FUNCTION_BLOCK PUBLIC FB_StationBase EXTENDS FB_ComponentBase IMPLEMENTS IStation
VAR_INPUT
	/// Enable items
	bEmergencyStopOk 	: BOOL;
	bSafetyOk 			: BOOL;
	bEnable 			: BOOL;
	bAutoHome 			: BOOL;		// if its true station will be homed by start button
	iNumberOfStepChains	: INT := 1;	// count of stepchains per station
	iStepChainIndex		: INT; 		// index to link text of choosed stepchain to hmi
END_VAR
VAR_OUTPUT
	nStateColor			: DWORD;	// color for state of station
	bBusy				: BOOL;		// station is busy
	bTransferEnable		: BOOL;		// transfer enable from station
	stTextAuto			: ST_Text;	// T_MaxString;
	stTextHome			: ST_Text;	// T_MaxString;
	
	/// error-stop status
	bAutoStop_Error		: BOOL;
END_VAR
VAR
	/// Refs
	stHmiToStation		: REFERENCE TO ST_DefaultHmiToPlc;				// default hmi to station
	stHmiManualIn		: REFERENCE TO ST_HMI_BASE_STATION_MANUAL_IN;	// hmi manual to station
	stHmiManualOut		: REFERENCE TO ST_HMI_BASE_STATION_MANUAL_OUT;	// hmi manual from station
	stLocalSettings		: REFERENCE TO ST_StationDynSettings;			// dyn. station settings
	stLocalMonitoring	: REFERENCE TO ST_Monitoring_Station;			// dyn. station monitoring
	
	stLocalSettingsBackup	: ST_StationDynSettings;	// dyn. station settings
	
	/// private var's
	nStationNb		: INT;
	eStation		: E_Station;
	eParent 		: E_Module;
	eOpMode			: E_OpMode;	
	bStopped		: BOOL := TRUE;
	bTipEnable		: BOOL;
	
	/// enable var's
	bRunCycle, bRunStep, 
	bRunHoming, bInHome,
	bEnableManualStep		 : BOOL;

	/// counter
	diCycles				: UDINT; // Zykluszähler
	diLastCycleTime			: UDINT; // letzte Zykluszeit [ms]
	
	tonOpModeOff			: TON;
	fTrigSafetyOk			: F_TRIG;
	rtrigOpModeChanged		: R_TRIG;
		
	rtirgSafetyOpMode_Auto	: R_TRIG;
	rtirgSafetyOpMode_Hand	: R_TRIG;
	rtirgSafetyOpMode_Aus	: R_TRIG;
	
	bInitSettings	: BOOL;
	bInitMonitoring	: BOOL;
	bInitManual		: BOOL;
	
	sb				: FB_StringBuilder;
	sqHome, sqAuto	: FB_SequenceHelperSb;
	localEvents		: ST_DefaultEventClasses;
END_VAR
VAR PERSISTENT
	diTotalCycles	: UDINT; // Zykluszähler
	eOpModeOld		: E_OpMode;
END_VAR

/// 
/// Station 01 function block 
///

{attribute 'monitoring' := 'call'}
PROPERTY Busy : BOOL
GET
Busy := bBusy;
END_GET
END_PROPERTY

METHOD PROTECTED CycleEnd
VAR_INPUT
END_VAR
diCycles := diCycles + 1;
diTotalCycles := diTotalCycles + 1;
diLastCycleTime := TIME_TO_UDINT(sqAuto.SeqTime);
sqAuto.StopSequence();
bBusy := FALSE;
bStopped := TRUE;
END_METHOD

{attribute 'monitoring':='call'}
PROPERTY PUBLIC Cycles : UDINT
GET
Cycles := diCycles;
END_GET
SET
diCycles := Cycles;
END_SET
END_PROPERTY

METHOD PROTECTED CycleStart
VAR_INPUT
END_VAR
sqAuto.StartSequence();
bBusy := TRUE;
bStopped := FALSE;
END_METHOD

{attribute 'monitoring':='call'}
PROPERTY PUBLIC EmergencyStopOk : BOOL
GET
EmergencyStopOk := bEmergencyStopOk;
END_GET
SET
bEmergencyStopOk := EmergencyStopOk;
END_SET
END_PROPERTY

{attribute 'monitoring':='call'}
PROPERTY PUBLIC Enable : BOOL
GET
Enable := bEnable;
END_GET
SET
bEnable := Enable;
END_SET
END_PROPERTY

{attribute 'monitoring':='call'}
//{attribute 'monitoring' := 'variable'}
PROPERTY PUBLIC EnableManual : BOOL
GET
EnableManual := EnableSummary AND (eOpMode = eOpMode_manual);
END_GET
END_PROPERTY

{attribute 'monitoring':='call'}
//{attribute 'monitoring' := 'variable'}
PROPERTY INTERNAL EnableSummary : BOOL
GET // PUBLIC
EnableSummary := bEnable 
				AND bSafetyOk 
				AND (bRunHoming OR (eOpMode = eOpMode_manual) OR (eOpMode = eOpMode_step) OR (eOpMode = eOpMode_auto));
END_GET
END_PROPERTY

METHOD PROTECTED GetComponentError : I_StringBuilder
VAR_IN_OUT
	fbUi	: FB_ManualUiBase;
END_VAR
VAR
	tmp		: ST_Text;
	name,
	err, 
	bmk		: STRING;
END_VAR
WSTRING_TO_STRING2(ADR(name), ADR(fbUi.stName.wsName), SIZEOF(name));		//ToDo: get rid of wstring?
WSTRING_TO_STRING2(ADR(err), ADR(fbUi.stErrorText.wsName), SIZEOF(err));
WSTRING_TO_STRING2(ADR(bmk), ADR(fbUi.stBmk.wsName), SIZEOF(bmk));

GetComponentError := sb.Set(name)
  .Append(' | ')  
  .Append(err)
  .Append(' | ')
  .Append(bmk);
END_METHOD

METHOD PUBLIC GetStepChainTest : ST_Text
VAR_INPUT
	Index : INT; // step chain index
END_VAR
// step chain index is ignored in the default implementation -> if multiple step chains are needed, use derived base and override this method. 
GetStepChainTest.nNameId := sqAuto.InfoTextId;
GetStepChainTest.wsName := sqAuto.Info.ToWString();
GetStepChainTest.wsNameId := sqAuto.InfoTextWsId;
END_METHOD

{attribute 'monitoring':='call'}
PROPERTY PUBLIC Homing : BOOL
GET
Homing := bRunHoming;
END_GET
END_PROPERTY

/// Station in Home flag
{attribute 'monitoring':='call'}
PROPERTY InHome : BOOL
GET
InHome := TRUE;
//FOR ii := 0 TO iNumberOfStepChains - 1 DO
	IF NOT sqHome.InHome THEN
		InHome := FALSE;
	END_IF
//END_FOR

bInHome := InHome;
IF InHome THEN
	bRunHoming := FALSE;
END_IF
END_GET
END_PROPERTY

METHOD PUBLIC InitEvents : IStation
VAR_IN_OUT CONSTANT
	infoEvent,
	warnEvent,
	errorEvent : TcEventEntry;
END_VAR
// create default station alarms
localEvents.Info := infoEvent;
localEvents.Warning := warnEvent;
localEvents.Error := errorEvent;
IEvent.CreateAlarm(infoEvent, FALSE, TcSourceInfo)
	  .CreateAlarm(warnEvent, TRUE, TcSourceInfo)
	  .CreateAlarm(errorEvent, TRUE, TcSourceInfo);

InitEvents := THIS^;
END_METHOD

METHOD PROTECTED M_CallObjects : BOOL
VAR_INPUT
END_VAR
// Call objects - to be subclassed
END_METHOD

METHOD PROTECTED M_DynMonitoring : BOOL
VAR_INPUT
END_VAR
// station base signals
stLocalMonitoring.bInHome := bInHome;
stLocalMonitoring.bAuto := bRunStep;
stLocalMonitoring.bBusy := bBusy;
stLocalMonitoring.bError := (eState = E_ComponentState.eComponentState_error);
stLocalMonitoring.bManual := (eOpMode = E_OpMode.eOpMode_manual);
stLocalMonitoring.bTransferEnable := bTransferEnable;
stLocalMonitoring.bWarning := (eState = E_ComponentState.eComponentState_warning);

M_DynMonitoring := TRUE;
END_METHOD

METHOD PUBLIC M_EnableSummary : BOOL
VAR_INPUT
END_VAR
END_METHOD

METHOD PROTECTED M_Homing
VAR
END_VAR
// Homing sequence - to be subclassed
END_METHOD

METHOD PUBLIC M_Init : IStation
VAR_INPUT
END_VAR
// set up defaults
Active := TRUE;
Enable := TRUE;
SUPER^.M_InitComponentBase();

// set up station id and name -> to be subclassed... 
//Station := E_Station.eStation_none;
//stName := stTextListGlobal.stText_ST000_Name;

sqAuto.SetInfo(Name);
nStateColor := TO_DWORD(STATICS.stColor.White);

stHmiToStation REF= P_HMI_Controller.aStHmiToStation[eStation];
stHmiManualIn REF= HMI.stHmi.stIn.arrStStation[eStation].stManual;
stHmiManualOut REF= HMI.stHmi.stOut.stCommon.arrStStation[eStation].stManual;
stLocalSettings REF= Services.stSettings.stStationSettings[eStation];
stLocalMonitoring REF= HMI.stHmi.stOut.stCommon.stMonitoring.astMonitoringStation[eStation];

//FOR ii := 0 TO CONST.iMaxIdxLocalStepChain DO
	sqAuto.SetInfo(stTextListGlobal.stText_initialize_station);	// -> to be subclassed, ... 
//END_FOR

M_Init := THIS^;
END_METHOD

METHOD PROTECTED M_InitDynManual : BOOL
VAR_INPUT
	nIndex			: INT;
	stName			: ST_Text;
	stGroup			: ST_Text;
	stType			: ST_Text;
	diObjectIndex	: DINT;
END_VAR
// chk
IF nIndex < 0 OR nIndex > CONST.iMaxIdxObject THEN
	StationError.ArgSbAppendRaise('Dyn. manual index out of range.');
	RETURN;
END_IF

stHmiManualOut.stObjects[nIndex].stName := stName;
stHmiManualOut.stObjects[nIndex].stGroup := stGroup;
stHmiManualOut.stObjects[nIndex].stType := stType;
stHmiManualOut.stObjects[nIndex].diObjectIndex := diObjectIndex;

M_InitDynManual := TRUE;
END_METHOD

METHOD PROTECTED M_InitDynManualUi : BOOL
VAR_IN_OUT
	fbManualUi	: FB_ManualUiBase;
END_VAR
VAR
	IManualUi	: I_ManualUi;
	nIx, ix		: INT;
END_VAR
IManualUi := fbManualUi;

// search next free index
nIx := -1;
FOR ix := 0 TO CONST.iMaxIdxObject DO
	IF stHmiManualOut.stObjects[ix].stName.wsName = "" THEN
		nIx := ix;
		EXIT;
	END_IF
END_FOR

IF nIx < 0 THEN
	StationError.ArgSbAppendRaise('Next free dyn. manual index not found.');
	RETURN;
END_IF

IManualUi.ObjectIndex := (StationNb * 1000) + nIx + 1; // create unique object index

M_InitDynManualUi := M_InitDynManual(nIx,			// index 
		IManualUi.Name,								// device name
		Name,										// group -> station name
		stTextListGlobal.stText_ObjectTypeDrive,	// type
		IManualUi.ObjectIndex);						// object index
		
IManualUi.M_SetStateObject(stHmiManualOut.stObjects[nIx]);
END_METHOD

METHOD PROTECTED M_InitDynMonitoringItem : BOOL
VAR_INPUT
	nIndex		: INT;
	wsName		: WSTRING;
	stGroup		: ST_Text;
	eDataType	: E_DataType;
	stUnit		: ST_Text;			
END_VAR
// chk
IF nIndex < 0 OR nIndex > CONST.iMaxIdxMonitoring THEN
	StationError.ArgSbAppendRaise('Dyn. monitoring index out of range.');
	RETURN;
END_IF

stLocalMonitoring.astMonitoring[nIndex].stIndex.nNameId := nIndex;
stLocalMonitoring.astMonitoring[nIndex].stIndex.wsNameId := wsName;
stLocalMonitoring.astMonitoring[nIndex].stName := F_CreateDynText(wsName, nIndex);
stLocalMonitoring.astMonitoring[nIndex].eDataType := eDataType;
stLocalMonitoring.astMonitoring[nIndex].stGroup := stGroup;
stLocalMonitoring.astMonitoring[nIndex].stUnit := stUnit;

M_InitDynMonitoringItem := TRUE;
END_METHOD

METHOD PROTECTED M_InitDynSettingsItem : BOOL
VAR_INPUT
	nIndex					: INT;
	wsIndex					: WSTRING;
	stSettGroup				: ST_Text;
	stSettTitle				: ST_Text;
	stSettUnit				: ST_Text;	
	eSettDataType			: E_DataType;	
	fSettValueMin			: REAL;
	fSettValueMax			: REAL;
	// required user level, 0 = none
	nRequiredUserLevel		: INT := 0;	
END_VAR
// chk
IF nIndex < 0 OR nIndex > CONST.iMaxIdxLocalSetting THEN
	StationError.ArgSbAppendRaise('Dyn. setting index out of range.');
	RETURN;
END_IF

M_InitDynSettingsItem := F_InitDynDataItem(
							nIndex,
							wsIndex,
							stSettGroup,
							stSettTitle,
							stSettUnit,
							eSettDataType,
							fSettValueMin,
							fSettValueMax,
							// required user level, 0 = none
							nRequiredUserLevel,
							E_RecipeMode.eRecipeMode_ToFrom,
							stLocalSettings.stDynStationSettings);
END_METHOD

METHOD PUBLIC M_InitEx : IStation
VAR_INPUT
	ILogger			: I_Logger;
	IEventHandler	: I_EventHandler;
END_VAR
M_InitEx := THIS^.M_Init();

// set up logger and event handler
SUPER^.M_InitComponentBaseEx(ILogger, IEventHandler);

// init extended stuff here...
END_METHOD

METHOD M_InitSequences : BOOL
VAR_INPUT
END_VAR
sqHome.Reset();
sqAuto.Reset(); 
sqAuto.SetInfo(stTextListGlobal.stText_initialize_station);
END_METHOD

METHOD PROTECTED M_Manual
VAR_INPUT
END_VAR
// Manual mode - to be subclassed
END_METHOD

METHOD PROTECTED M_OpModeChanged : BOOL
VAR_INPUT
END_VAR
// to be subclassed
END_METHOD

METHOD PUBLIC M_Run : BOOL
VAR
END_VAR
M_Run := TRUE; // to be subclassed..

// call component run
SUPER^.Run();

// Safety OP-Mode
rtirgSafetyOpMode_Auto(CLK := stHmiToStation.eSafetyOpMode = E_Opmode.eOpMode_auto);
rtirgSafetyOpMode_Hand(CLK := stHmiToStation.eSafetyOpMode = E_Opmode.eOpMode_manual);
rtirgSafetyOpMode_Aus(CLK := stHmiToStation.eSafetyOpMode = E_Opmode.eOpMode_off);

// reset (all or this station)
IF stHmiToStation.bReset THEN
	Reset();
END_IF

// step (all or this station)
// step -> ist bei Auto über die Property immer TRUE
bRunStep := stHmiToStation.bStep;
	
// start (all or this station)
IF stHmiToStation.bStart OR P_Safety.bMachineRequestStart OR stHmiToStation.bStep THEN		
	IF NOT bEnable THEN
		StationWarning.ArgSetString('Kein Enable Signal bei Start').Raise();
	ELSIF NOT bSafetyOk THEN
		StationWarning.ArgSetString('Safety nicht ok bei Start').Raise();
	// Fehler steht noch an
	ELSIF bAutoStop_Error THEN
		StationWarning.ArgSetString('Station in Fehlerstatus --> Reset').Raise();

	// Safety muss in Auto sein
	ELSIF stHmiToStation.eSafetyOpMode <> E_Opmode.eOpMode_auto AND Const.bEnSafetyOpMode THEN
		StationWarning.ArgSetString('Safety Betriebsart nicht AUTO').Raise();
		
	// START
	ELSIF (OpMode = E_Opmode.eOpMode_auto OR OpMode = E_Opmode.eOpMode_step) THEN
		//bRunStep := FALSE;
		bRunCycle := TRUE;
	END_IF
END_IF

// cycle stop (all or this station)
IF stHmiToStation.bStop OR P_Safety.bMachineRequestCycleStop OR P_Supervision.bCycleStop THEN
	bRunCycle := bRunHoming := FALSE;
END_IF

// fast stop (all or this station)
IF stHmiToStation.bFastStop OR P_Supervision.bFastStop THEN 
	bRunCycle := bRunStep := bRunHoming := FALSE;
END_IF

// set op mode (all or this station)
tonOpModeOff(IN := stHmiToStation.bStop, PT := T#10S);
IF stHmiToStation.bOpModeManual OR rtirgSafetyOpMode_Hand.Q THEN
	bRunStep := FALSE;
	bRunCycle := FALSE;
	bRunHoming := FALSE;
	eOpMode := E_OpMode.eOpMode_manual;
ELSIF stHmiToStation.bOpModeAuto OR rtirgSafetyOpMode_Auto.Q THEN
	bRunStep := FALSE;
	bRunCycle := FALSE;
	bRunHoming := FALSE;
	eOpMode := E_OpMode.eOpMode_auto;
ELSIF stHmiToStation.bOpModeStep THEN
	bRunStep := FALSE;
	bRunCycle := FALSE;
	bRunHoming := FALSE;
	eOpMode := E_OpMode.eOpMode_step;
ELSIF tonOpModeOff.Q THEN
	eOpMode := E_OpMode.eOpMode_off;
END_IF
	
IF NOT bEmergencyStopOk THEN
	sqHome.InHome := FALSE;
	sqHome.Step := 0;
	sqAuto.Step := 0;
END_IF

// homing (all or this station)
IF stHmiToStation.bHome OR (stHmiToStation.bStart AND bAutoHome AND NOT sqHome.InHome AND sqHome.Step = 0 AND sqAuto.Step = 0) THEN
	IF NOT bEnable THEN
		StationWarning.ArgSbAppendRaise('Kein Enable Signal bei Start Grundstellung');
	ELSIF NOT bSafetyOk THEN
		StationWarning.ArgSbAppendRaise('Safety nicht ok bei Start Grundstellung');
		
	// Fehler steht noch an
	ELSIF bAutoStop_Error THEN
		StationWarning.ArgSbAppendRaise('Station in Fehlerstatus --> Reset');
	ELSE		
		sqHome.Step := 0;
		sqHome.InHome		:= FALSE;
		bRunCycle			:= FALSE;
		bRunHoming 			:= TRUE;
	END_IF
END_IF

/// Set Station State Color
IF State = eComponentState_error THEN
	nStateColor := STATICS.stColor.Red;
ELSIF bInHome AND (eOpMode = eOpMode_Auto OR eOpMode = eOpMode_Step) THEN	
	nStateColor := STATICS.stColor.LightBlue;
ELSIF bStopped AND (eOpMode = eOpMode_Auto OR eOpMode = eOpMode_Step) THEN
	nStateColor := STATICS.stColor.Blue;									
ELSIF State = eComponentState_running AND (eOpMode = eOpMode_Auto OR eOpMode = eOpMode_Step) THEN
	nStateColor := STATICS.stColor.LimeGreen;					
ELSIF State = eComponentState_running AND eOpMode = eOpMode_manual THEN
	nStateColor := STATICS.stColor.Orange;		
ELSE
	nStateColor := STATICS.stColor.White;
END_IF

//StepChainTextMapping
//stTextAuto := arraSTextAuto[iStepChainIndex];
//IF iStepChainIndex >= 0 AND iStepChainIndex <= CONST.iMaxIdxLocalStepChain THEN
	stTextAuto.nNameId := sqAuto.InfoTextId;
	stTextAuto.wsName := WConcat3(TO_WSTRING(sqAuto.Step),": ", sqAuto.Info.ToWString());
	stTextAuto.wsNameId := WConcat3(TO_WSTRING(sqAuto.Step),": ", sqAuto.InfoTextWsId);	
	
	//stTextHome := arraSTextHome[iStepChainIndex];
	stTextHome.nNameId := sqHome.InfoTextId;
	stTextHome.wsName := WConcat3(TO_WSTRING(sqHome.Step), ": ", sqHome.Info.ToWString());
	stTextHome.wsNameId := WConcat3(TO_WSTRING(sqHome.Step),": ", sqHome.InfoTextWsId);
//END_IF

rtrigOpModeChanged(CLK := eOpModeOld <> eOpMode);
IF rtrigOpModeChanged.Q THEN
	eOpModeOld := eOpMode;
	M_OpModeChanged();
END_IF

//call methodes
sqHome.EnableStep := RunStep;
sqHome();
sqAuto.EnableStep := RunStep;
sqAuto();

M_CallObjects();
M_Homing();
M_Sequence();
M_Manual();
M_Supervision();
END_METHOD

METHOD PROTECTED M_Sequence
VAR
END_VAR
// Automatic sequence - to be subclassed
END_METHOD

METHOD PROTECTED M_Supervision : BOOL
VAR_INPUT
END_VAR
// to be subclassed
END_METHOD

/// Station OP Mode
{attribute 'monitoring':='call'}
PROPERTY OpMode : E_OpMode
GET
OpMode := eOpMode;
END_GET
END_PROPERTY

{attribute 'monitoring':='call'}
PROPERTY Parent : E_Module
GET
Parent := eParent;
END_GET
END_PROPERTY

METHOD PROTECTED ReactToComponentError
VAR_IN_OUT
	fbUi	: FB_ManualUiBase;
END_VAR
VAR_INPUT
	mode 	: E_EventReaction;
END_VAR
VAR
	msg		: I_StringBuilder;
END_VAR
msg := GetComponentError(fbUi);
ReactToEvent(mode, TcEventSeverity.Error)
			.ArgSetSbRaise(msg);
END_METHOD

METHOD PROTECTED ReactToError : I_EventHandler
VAR_INPUT
	mode : E_EventReaction;
END_VAR
ReactToError := ReactToEvent(mode, TcEventSeverity.Error);
END_METHOD

METHOD PROTECTED ReactToEvent : I_EventHandler
VAR_INPUT
	mode		: E_EventReaction;
	severity	: TcEventSeverity;
END_VAR
// switch event reaction mode
CASE mode OF
	E_EventReaction.Init:
		M_InitSequences();
		
	E_EventReaction.Stop:
		bRunCycle := FALSE;
		bAutoStop_Error := TRUE;
		
	E_EventReaction.CycleStop:
		bRunCycle := FALSE;
		
END_CASE

// set the component state &
//  return value (info, warning or error - event handler)
CASE severity OF
	TcEventSeverity.Info:
		eState := E_ComponentState.eComponentState_info;
		ReactToEvent := StationInfo;
		
	TcEventSeverity.Warning:
		eState := E_ComponentState.eComponentState_warning;
		ReactToEvent := StationWarning;
		
	ELSE
		eState := E_ComponentState.eComponentState_error;
		ReactToEvent := StationError;
		
END_CASE
END_METHOD

METHOD PROTECTED ReactToInfo : I_EventHandler
VAR_INPUT
	mode : E_EventReaction;
END_VAR
ReactToInfo := ReactToEvent(mode, TcEventSeverity.Info);
END_METHOD

METHOD PROTECTED ReactToWarn : I_EventHandler
VAR_INPUT
	mode : E_EventReaction;
END_VAR
ReactToWarn := ReactToEvent(mode, TcEventSeverity.Warning);
END_METHOD

/// Reset component logic
{attribute 'object_name' := 'Reset'}
METHOD Reset
VAR
	iIdxSub			: INT;
END_VAR
// base logic run
SUPER^.Reset();

// reset var's
nStateColor := STATICS.stColor.White;

bAutoStop_Error := FALSE;
END_METHOD

{attribute 'monitoring':='call'}
PROPERTY PUBLIC RunCycle : BOOL
GET // PUBLIC
RunCycle := bRunCycle;
END_GET
SET // PUBLIC
bRunCycle := RunCycle;
END_SET
END_PROPERTY

{attribute 'monitoring':='variable'}
PROPERTY PUBLIC RunManStep : Bool
GET
RunManStep := EnableSummary AND
			NOT bAutoStop_Error AND
			(OpMode = E_OpMode.eOpMode_manual AND (bRunStep OR NOT bEnableManualStep));
END_GET
END_PROPERTY

{attribute 'monitoring':='variable'}
PROPERTY PUBLIC RunStep : BOOL
GET
VAR
	sMsg : WSTRING(255);
END_VAR
// Rückgabe
RunStep := EnableSummary AND
			NOT bAutoStop_Error AND
			((bRunStep AND eOpMode = eOpMode_step) OR
			(eOpMode = eOpMode_auto));
END_GET
END_PROPERTY

{attribute 'monitoring':='call'}
PROPERTY PUBLIC SafetyOk : BOOL
GET
SafetyOk := bSafetyOk;
END_GET
SET
bSafetyOk := SafetyOk;
END_SET
END_PROPERTY

{attribute 'monitoring':='call'}
PROPERTY StateColor : DWORD
GET
StateColor := nStateColor;
END_GET
END_PROPERTY

{attribute 'monitoring':='call'}
PROPERTY PUBLIC Station : E_Station
GET
Station := eStation;
END_GET
SET // PUBLIC
eStation := Station;
END_SET
END_PROPERTY

PROPERTY PROTECTED StationError : I_EventHandler
GET
// return the event handler
//	prepare string builder w. station info
StationError := IEvent.Select(localEvents.Error)
					  .ArgSbInitWs(stName.wsName)
					  .ArgSbAppend(' | ');
END_GET
END_PROPERTY

PROPERTY PROTECTED StationInfo : I_EventHandler
GET
// return the event handler
//	prepare string builder w. station info
StationInfo := IEvent.Select(localEvents.Info)
					 .ArgSbInitWs(stName.wsName)
					 .ArgSbAppend(' | ');
END_GET
END_PROPERTY

PROPERTY PUBLIC StationNb : INT
GET
StationNb := nStationNb;
END_GET
SET // PUBLIC
nStationNb := StationNb;
END_SET
END_PROPERTY

PROPERTY PROTECTED StationWarning : I_EventHandler
GET
// return the event handler
//	prepare string builder w. station info
StationWarning := IEvent.Select(localEvents.Warning)
					 .ArgSbInitWs(stName.wsName)
					 .ArgSbAppend(' | ');
END_GET
END_PROPERTY

/// Station stopped
{attribute 'monitoring':='call'}
PROPERTY Stopped : BOOL
GET
Stopped := bStopped;
END_GET
END_PROPERTY

PROPERTY TextAuto : ST_Text
GET
TextAuto := stTextAuto;
END_GET
END_PROPERTY

PROPERTY TextHome : ST_Text
GET
TextHome := stTextHome;
END_GET
END_PROPERTY

{attribute 'monitoring':='call'}
PROPERTY PUBLIC TipEnable : BOOL
GET
TipEnable := bTipEnable;
END_GET
END_PROPERTY

{attribute 'monitoring':='call'}
PROPERTY PUBLIC TotalCycles : UDINT
GET
TotalCycles := diTotalCycles;
END_GET
END_PROPERTY

{attribute 'monitoring' := 'call'}
PROPERTY TransferEnable : BOOL
GET
TransferEnable := bTransferEnable;
END_GET
END_PROPERTY

END_FUNCTION_BLOCK

(* stored: Version 1.1.0.1
   POU FB_StationBase: Id {f54fb284-2edb-421a-b9be-72585b0b821e}, SpecialFunc None
   Folder DynSetMonMan: Id {9deb34dc-1f16-478f-962a-d4d1b0f552c1}
   Folder Events: Id {027c7c1e-e36c-4140-af0c-88182745993a}
   Folder Internal: Id {94411a46-819e-4d59-aec8-167df78a8a36}
   Folder Properties: Id {b426106f-419d-411b-b553-37fa2c35c33a}
   Folder Protected: Id {c662f486-9e5e-4c19-88f4-4fa8c599a7ba}
   Property Busy: Id {8819031e-05ae-422b-bdb7-78b68817a347}
   Get Get: Id {c3d1589d-72fb-476f-9581-5e78d8c51428}
   Method CycleEnd: Id {42e03c24-27ed-48e3-8ed0-281947e6589c}
   Property Cycles: Id {72db52e1-d2fe-44b2-a519-b0c67b5de69f}
   Get Get: Id {f79db9f1-0039-405b-9fde-7f22d9ed7f0d}
   Set Set: Id {c7a50d01-0ad3-48e2-a41a-d38e4b0da7e3}
   Method CycleStart: Id {333997de-eae7-46e7-8371-d8e2ed4c4b92}
   Property EmergencyStopOk: Id {5a59110c-785a-45ad-a350-85d44acaa434}
   Get Get: Id {f0423ab1-f2df-419a-8af2-5ca45ca5a78d}
   Set Set: Id {e2b7c6a7-9d09-457a-b825-4bd298996c19}
   Property Enable: Id {28347798-46db-4e64-8ab3-4ee921f419e1}
   Get Get: Id {204cb216-e414-441d-9e8d-b48ebcf1d619}
   Set Set: Id {20a0bb48-9a2c-4453-ac04-ad07ff2ceb1b}
   Property EnableManual: Id {94bc03c1-c1c5-49bf-a2b7-cf6f0f61c0c7}
   Get Get: Id {a50db3e9-109a-4814-a3ca-6b9f7ee02a81}
   Property EnableSummary: Id {d38cad44-3c6b-473e-9228-06674de6bb5c}
   Get Get: Id {b84f63c5-1a72-4487-a1fa-3c5260569776}
   Method GetComponentError: Id {e291252f-0029-41c9-9cac-3999e02b4e3d}
   Method GetStepChainTest: Id {6b5c222a-2357-4c9b-9bbd-ad1c2653fe0f}
   Property Homing: Id {ff9f0f9c-0627-4634-97ff-526f2aca4a5e}
   Get Get: Id {992234dc-a116-4c9a-9cb6-2d39c89e14a3}
   Property InHome: Id {6a5ace07-5006-4caa-b686-c8b542cb3a49}
   Get Get: Id {620ea1cd-6ef3-450e-8e8d-d7e211d4ad3c}
   Method InitEvents: Id {f7ca0fb6-bc90-4005-9d7e-929db98cbd24}
   Method M_CallObjects: Id {9fe3b799-e5c7-4b43-9648-840569809409}
   Method M_DynMonitoring: Id {dfe69796-4aec-4952-ad4d-ff3543df6a88}
   Method M_EnableSummary: Id {65c2d347-9b3e-4a50-ba8b-e531af5e016d}
   Method M_Homing: Id {af9cad83-ca55-4385-a049-15fbacdc5a5f}
   Method M_Init: Id {dd195e2f-de60-4c36-b80c-fe91574eb32b}
   Method M_InitDynManual: Id {694f5279-f539-4db9-a107-1ad97e411fbb}
   Method M_InitDynManualUi: Id {a093ea62-0ed7-43f2-9d3d-c205c0028916}
   Method M_InitDynMonitoringItem: Id {75c32d60-2a6d-4406-a748-73d378a60d34}
   Method M_InitDynSettingsItem: Id {c58a2340-e337-4ec5-b5c0-cb90b5f97eba}
   Method M_InitEx: Id {ee927414-04b1-467a-ae4b-7b83ebf46dd2}
   Method M_InitSequences: Id {0857e067-a4a3-4623-ba2f-3f66c5028e4a}
   Method M_Manual: Id {431a609a-f059-457f-8f7c-6f6273bdcc5d}
   Method M_OpModeChanged: Id {78264e7c-3b2e-4bf7-8226-a0400a0094f3}
   Method M_Run: Id {4bea32ab-ef45-430f-b1b8-b1769c0ad78d}
   Method M_Sequence: Id {bde17e20-9713-4c0f-bbf7-0898047c9be7}
   Method M_Supervision: Id {9514cef4-a5c0-43d3-a29b-3106f77c8bdb}
   Property OpMode: Id {6d3f4baa-a078-4b2d-8d0c-5708af5427ae}
   Get Get: Id {f47e60fe-3e52-4086-9cde-a02b5212fd56}
   Property Parent: Id {c5e1ee97-3992-4724-87a8-cb2744aa19d4}
   Get Get: Id {3309f75f-9fc0-43fc-af3e-44eb4101d093}
   Method ReactToComponentError: Id {1e078b5b-c346-4292-b9cd-2516432a2b86}
   Method ReactToError: Id {070a1f6d-05e9-4ac5-b65c-0cb42b813665}
   Method ReactToEvent: Id {101b3096-47b5-4e81-bda7-e9ab65e8f446}
   Method ReactToInfo: Id {67241799-906c-49ef-8ba4-9bbdffe4afa7}
   Method ReactToWarn: Id {e962099f-315e-4997-b2ec-93b2afa00f53}
   Method Reset: Id {5f70ca86-af08-4351-9508-32c132c3c4ee}
   Property RunCycle: Id {4ecb12c0-ab26-460b-9508-2a31719ab90f}
   Get Get: Id {fa7d0a0e-ce19-4870-b288-7d4a50ef6e28}
   Set Set: Id {751a28e8-91e1-46e5-a197-9b0c0ef27836}
   Property RunManStep: Id {bebf9843-2bf1-4211-9e43-ad5dcf762cbe}
   Get Get: Id {b3a7a39c-b06b-40c8-9401-97baca3fa651}
   Property RunStep: Id {2cd1a20d-9c63-48a7-aef5-2e9908460bef}
   Get Get: Id {9386ea9e-764e-4c1a-9ce1-22eaa413ff55}
   Property SafetyOk: Id {a67c08f6-8ad4-4d81-a010-3913e3bd7238}
   Get Get: Id {3da21f09-1d7a-46ea-9ffa-41ed50561650}
   Set Set: Id {a93c8863-f6f4-4850-b6ca-51f22cdb652e}
   Property StateColor: Id {687b22f0-0e68-427b-a85a-0302eb703e69}
   Get Get: Id {e9616a59-e72f-4d0e-ad21-267c11b87e1c}
   Property Station: Id {7931aaf1-8e2e-475b-b475-068cd1ac9a70}
   Get Get: Id {46b6a482-e32f-4499-87aa-fe521bb5e07b}
   Set Set: Id {3556564d-f5fd-4ce5-95ed-c554ddaa9077}
   Property StationError: Id {2b2f8078-2002-44cd-b9fe-a71886e893d2}
   Get Get: Id {af7c6bd2-d919-44f8-8205-c22b25515ef2}
   Property StationInfo: Id {c46898e7-5389-4291-b5b5-532e2be10697}
   Get Get: Id {58eac9b2-e4fb-4a16-a00d-87f9f31d5dd6}
   Property StationNb: Id {ef929b85-9b28-4e1d-b2fb-66c6c26d4c85}
   Get Get: Id {4a4ea237-3bf9-4723-ad34-60b96c4d5da0}
   Set Set: Id {d96e1c9d-5c50-41ce-ac73-f96520a69f47}
   Property StationWarning: Id {6f1898b6-e230-495d-ad79-e2373ed4df1b}
   Get Get: Id {f6d49f2f-6d1d-4d8e-b736-afe2aee54775}
   Property Stopped: Id {49c76449-1083-494a-9050-1b4ec6c6ad7b}
   Get Get: Id {d3b09b7a-a47f-4359-92d3-333447cf649a}
   Property TextAuto: Id {625841f2-a00b-4d0e-b750-e833d3fe1cca}
   Get Get: Id {85557adc-355a-41ec-a98d-2426d5ddda20}
   Property TextHome: Id {a7c5efda-84c2-4055-a17c-84a3db4aa14e}
   Get Get: Id {6d69fad5-2116-4db7-b85d-bef54ce60c33}
   Property TipEnable: Id {e7f11a41-affb-4d8e-b05a-b3c91ed6b314}
   Get Get: Id {847d006c-2c56-482e-862a-eeae3c6ef6c0}
   Property TotalCycles: Id {3ee925cd-a881-48f1-94ac-01ecc529e277}
   Get Get: Id {7ab5f762-41b4-4ee7-bc77-bfe675622cac}
   Property TransferEnable: Id {7653d16a-7b93-441f-87bb-66fbf54f407e}
   Get Get: Id {d06abcfc-d96c-4059-8ae9-065f5dbc17a6} *)
